FUNCTION_BLOCK ConveyorCTLCentralClient (* Basic Function Block Type *)
  (* Standard: 61499-2 *)
  (* Version 0.2, 2003-12-04, JHC, Rockwell Automation, Renamed for better indexing. *)
  (* Version 0.1, 2002-11-05, JHC, Rockwell Automation, Corrected missing ST element in Algorithm REQ. *)
  (* Version 0.0, 2000-05-30, JHC, Rockwell Automation *)
  (* Compiler header: package fb.rt.cs725; *)
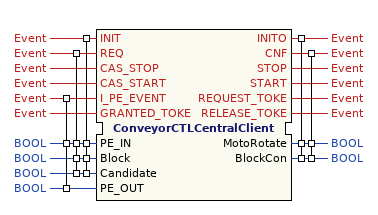
  EVENT_INPUT
    INIT WITH PE_IN, Block, Candidate; (* Initialization Request *)
    REQ WITH PE_IN, Block, Candidate; (* Normal Execution Request *)
    CAS_STOP;
    CAS_START;
    I_PE_EVENT WITH PE_IN, PE_OUT;
    GRANTED_TOKE;
  END_EVENT
  EVENT_OUTPUT
    INITO WITH MotoRotate, BlockCon; (* Initialization Confirm *)
    CNF WITH MotoRotate, BlockCon; (* Execution Confirmation *)
    STOP;
    START;
    REQUEST_TOKE;
    RELEASE_TOKE;
  END_EVENT
  VAR_INPUT
    PE_IN : BOOL; (* Input event qualifier *)
    Block : BOOL;
    Candidate : BOOL;
    PE_OUT : BOOL; (* Output event qualifier *)
  END_VAR
  VAR_OUTPUT
    MotoRotate : BOOL; (* Output event qualifier *)
    BlockCon : BOOL;
  END_VAR
  VAR
    lastPE : BOOL := 1;
    lastBlock : BOOL := 0;
  END_VAR
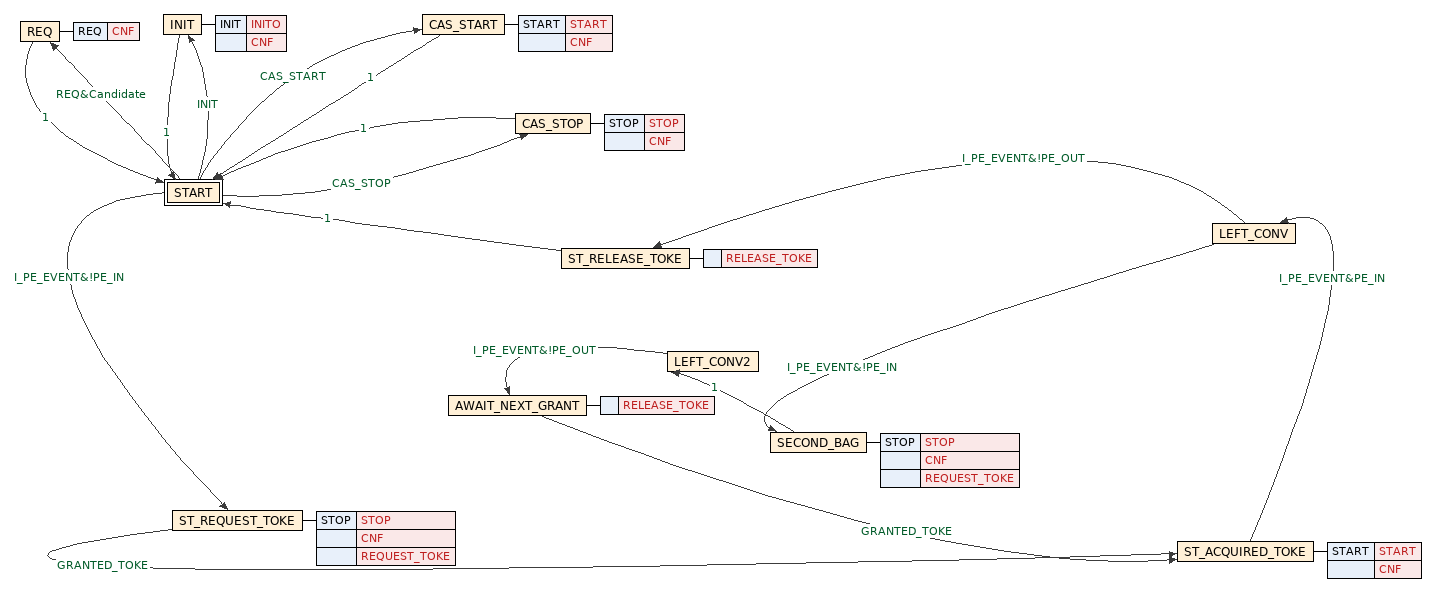
  EC_STATES
    START; (* Initial State *)
    INIT : INIT -> INITO, -> CNF; (* Initialization *)
    REQ : REQ -> CNF; (* Normal execution *)
    CAS_START : START -> START, -> CNF;
    CAS_STOP : STOP -> STOP, -> CNF;
    ST_REQUEST_TOKE : STOP -> STOP, -> CNF, -> REQUEST_TOKE;
    ST_ACQUIRED_TOKE : START -> START, -> CNF;
    ST_RELEASE_TOKE : -> RELEASE_TOKE;
    LEFT_CONV;
    SECOND_BAG : STOP -> STOP, -> CNF, -> REQUEST_TOKE;
    LEFT_CONV2;
    AWAIT_NEXT_GRANT : -> RELEASE_TOKE;
  END_STATES
  EC_TRANSITIONS
    START TO INIT := INIT;
    INIT TO START := 1;
    START TO REQ := REQ&Candidate;
    REQ TO START := 1;
    START TO CAS_START := CAS_START;
    CAS_START TO START := 1;
    START TO CAS_STOP := CAS_STOP;
    CAS_STOP TO START := 1;
    ST_RELEASE_TOKE TO START := 1;
    LEFT_CONV TO ST_RELEASE_TOKE := I_PE_EVENT&!PE_OUT;
    ST_ACQUIRED_TOKE TO LEFT_CONV := I_PE_EVENT&PE_IN;
    START TO ST_REQUEST_TOKE := I_PE_EVENT&!PE_IN;
    LEFT_CONV TO SECOND_BAG := I_PE_EVENT&!PE_IN;
    SECOND_BAG TO LEFT_CONV2 := 1;
    ST_REQUEST_TOKE TO ST_ACQUIRED_TOKE := GRANTED_TOKE;
    LEFT_CONV2 TO AWAIT_NEXT_GRANT := I_PE_EVENT&!PE_OUT;
    AWAIT_NEXT_GRANT TO ST_ACQUIRED_TOKE := GRANTED_TOKE;
  END_TRANSITIONS
  ALGORITHM INIT IN ST: (* Initialization algorithm *)
MotoRotate := TRUE;
Block := FALSE;

System.out.println(this + " " + MotoRotate);
System.out.println(MotoRotate);
  END_ALGORITHM
  ALGORITHM REQ IN ST: (* Normally executed algorithm *)
System.out.println(this +  " -> Candidate" + Candidate);
IF Candidate THEN
IF lastPE !:= PE_IN THEN
IF NOT PE_IN THEN
BlockCon:= TRUE;
System.out.println("BlockCon = true");
ELSE
BlockCon:=FALSE;
System.out.println("BlockCon = false");
END_IF
lastPE := PE_IN;
END_IF
IF lastBlock !:= Block THEN
IF Block THEN
STOP.serviceEvent(this);
MotoRotate := FALSE;
System.out.println("Cas Stop");
ELSE
START.serviceEvent(this);
MotoRotate := TRUE;
System.out.println("Cas Start");
END_IF
lastBlock := Block;
END_IF
END_IF
  END_ALGORITHM
  ALGORITHM START IN ST:
MotoRotate:=TRUE;
System.out.println(this + " Start " + MotoRotate);

System.out.println("Start " + MotoRotate);
  END_ALGORITHM
  ALGORITHM STOP IN ST:
MotoRotate := FALSE;
System.out.println(this + " Stop " + MotoRotate);

System.out.println("Stop " + MotoRotate);
  END_ALGORITHM
END_FUNCTION_BLOCK
